FUNCTION_BLOCK fb_eventController
VAR_INPUT
in_flg_run : BOOL;
END_VAR
VAR_OUTPUT
	out_flg_run : BOOL;
END_VAR
VAR

	fbi_eventListGenerator: ARRAY [0..50] OF fb_eventListGenerator;
	var_semaphore: INT;
	var_alarmQty: INT;
	flg_errorTrg: ARRAY[0..50] OF BOOL;

    var_timeAsDT : DT;
	var_alarmListLog: s_alarmList;
	flg_reqUpdate: BOOL;
	fbi_r_TRIG: R_TRIG;
	var_n: INT;
	fbi_buzzerGenerater: fb_buzzerGenerater;
	var_n2: INT;
	var_alarmListEmpty : s_alarmList;
	fbi_GetLocalAmsNetId: FB_GetLocalAmsNetId;
	fbi_LocalSystemTime: FB_LocalSystemTime;
	fbi_ton1: TON;
	var_i: INT;
	fbi_first: TON;
	var_dummy: ARRAY [1..10] OF s_str_alarmList;
END_VAR
VAR_STAT
	flg_error: BOOL;
	flg_warning: BOOL;
	flg_info: BOOL;
END_VAR
VAR // added by the converter: edge detectors and wires of the graphical bodies
    _rt1 : R_TRIG;
END_VAR

eventList();

//get current time
fbi_GetLocalAmsNetId(
	bExecute:=TRUE , 
	tTimeOut:= ,
	bBusy=> , 
	bError=> , 
	nErrId=> , 
	AddrString=> , 
	AddrBytes=> );


fbi_LocalSystemTime(
	sNetID:=fbi_GetLocalAmsNetId.AddrString , 
	bEnable:= TRUE, 
	dwCycle:= , 
	dwOpt:= , 
	tTimeout:= , 
	bValid=> , 
	systemTime=> , 
	tzID=> );

var_timeAsDT := SYSTEMTIME_TO_DT(fbi_LocalSystemTime.systemTime);
//reset

//
IF gvl_error.flg_error THEN
	gvl_error.flg_alramBusy := TRUE;
END_IF

fbi_r_TRIG(CLK:= flg_requpdate, Q=> );
//event log update
IF fbi_r_TRIG.Q THEN
	FOR var_n := 50 TO 2 BY -1 DO
			gvl_error.var_ary_alarmlistLog[var_n].var_alarmName := gvl_error.var_ary_alarmlistLog[var_n-1].var_alarmName;
			gvl_error.var_ary_alarmlistLog[var_n].var_alarmLevel := gvl_error.var_ary_alarmlistLog[var_n-1].var_alarmLevel;
			gvl_error.var_ary_alarmlistLog[var_n].var_alarmMassge := gvl_error.var_ary_alarmlistLog[var_n-1].var_alarmMassge;
			gvl_error.var_ary_alarmlistLog[var_n].var_alarmTime := gvl_error.var_ary_alarmlistLog[var_n-1].var_alarmTime;
			gvl_error.var_ary_alarmlistLog[var_n].var_alarmCode1 := gvl_error.var_ary_alarmlistLog[var_n-1].var_alarmCode1;
			gvl_error.var_ary_alarmlistLog[var_n].var_alarmCode2 := gvl_error.var_ary_alarmlistLog[var_n-1].var_alarmCode2;
			
			IF var_n = 2 THEN
				gvl_error.var_ary_alarmlistLog[1].var_alarmName := var_alarmListLog.var_alarmName;
				gvl_error.var_ary_alarmlistLog[1].var_alarmLevel := var_alarmListLog.var_alarmLevel;
				gvl_error.var_ary_alarmlistLog[1].var_alarmMassge := var_alarmListLog.var_alarmMassge;
				gvl_error.var_ary_alarmlistLog[1].var_alarmTime := var_alarmListLog.var_alarmTime;
				gvl_error.var_ary_alarmlistLog[1].var_alarmCode1 := var_alarmListLog.var_alarmCode1;
				gvl_error.var_ary_alarmlistLog[1].var_alarmCode2 := var_alarmListLog.var_alarmCode2;
				var_semaphore := var_semaphore - 1;
			END_IF
		END_FOR	
END_IF

//reset realtime event 
IF gvl_error.flg_eventDisplayRest THEN
	FOR var_n2 := 1 TO 10 BY 1 DO
		gvl_error.var_ary_alarmlistActive[var_n2].var_alarmCode1 := eP_alarmCode._;
		gvl_error.var_ary_alarmlistActive[var_n2].var_alarmCode2 := '';
		gvl_error.var_ary_alarmlistActive[var_n2].var_alarmLevel := '';
		gvl_error.var_ary_alarmlistActive[var_n2].var_alarmMassge := "";
		gvl_error.var_ary_alarmlistActive[var_n2].var_alarmName := "";
		gvl_error.var_ary_alarmlistActive[var_n2].var_alarmTime := '';
	END_FOR
END_IF
//massage
	flg_info := gvl_error.flg_warning OR gvl_error.flg_info OR gvl_error.flg_sample_windown_warning;
	IF NOT flg_info THEN
		gvl_visu.var_msg := "";	
	END_IF
//buzzer
fbi_buzzerGenerater(
	in_flg_LvError:=gvl_error.flg_error OR gvl_error.flg_sample_windown_warning,
	in_flg_LvWarning:=gvl_error.flg_warning,
	in_flg_LvInfo:=gvl_error.flg_info ,
	out_flg_buzzer=> gvl_io.flg_signalTowerBuzzer ,
	out_flg_Yellow=> gvl_io.flg_signalTowerYellow
);
gvl_io.flg_signalTowerRed := gvl_error.flg_error;

IF gvl_error.flg_ararmLevelRest THEN
	gvl_error.flg_error := FALSE;
	gvl_error.flg_warning := FALSE;
	gvl_error.flg_info := FALSE;
END_IF

ACTION eventList:
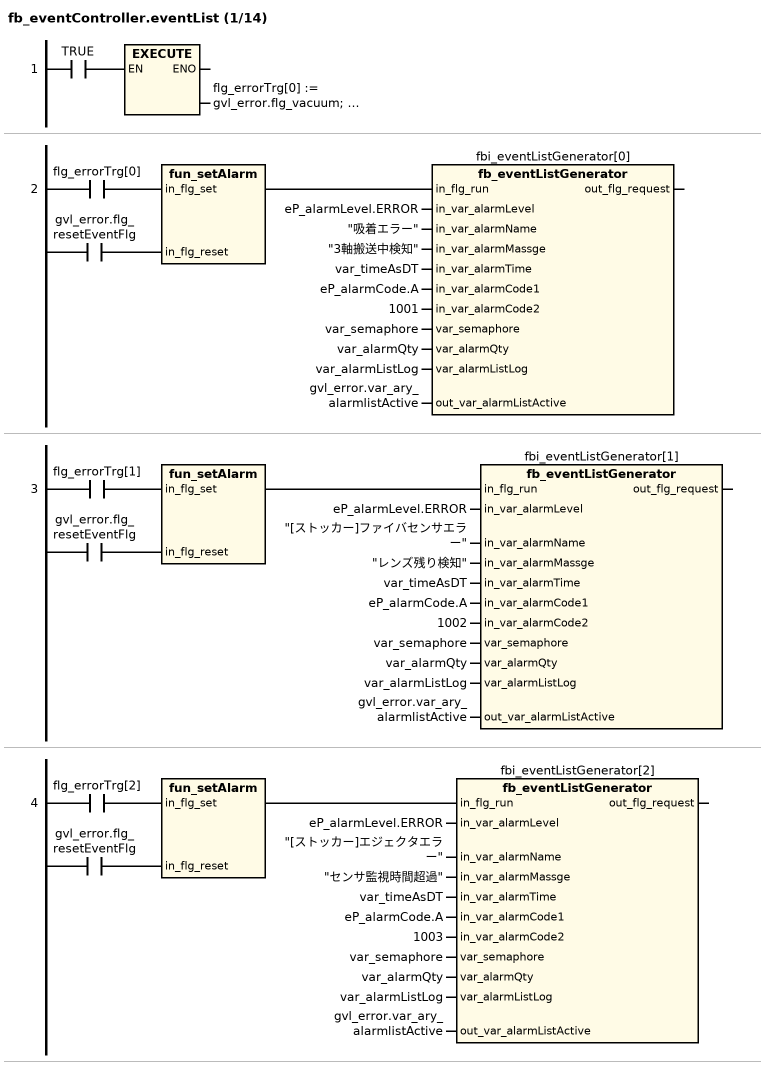
// NETWORK 1
flg_errorTrg[0] := gvl_error.flg_vacuum;
flg_errorTrg[1] := gvl_error.flg_fiberSens;
flg_errorTrg[2] := gvl_solv.fbi_ejector.out_flg_error;
flg_errorTrg[3] := gvl_solv.fbi_chuck.out_flg_error;
flg_errorTrg[4] := gvl_solv.fbi_push.out_flg_error;
flg_errorTrg[5] := gvl_elecylinder.fbi_axisTransport.out_flg_error;
flg_errorTrg[6] := gvl_elecylinder.fbi_axisSample.out_flg_error;
flg_errorTrg[7] := gvl_elecylinder.fbi_axisTrayChange.out_flg_error OR gvl_error.flg_trayChangeError;
flg_errorTrg[8] := gvl_elecylinder.ref_axis_transport.input.in_wire_error;
flg_errorTrg[9] := gvl_elecylinder.ref_axis_sample.input.in_wire_error;
flg_errorTrg[10] := gvl_elecylinder.ref_axis_trayChange.input.in_wire_error;
flg_errorTrg[11] := gvl_axis.ref_x.Error;
flg_errorTrg[12] := gvl_axis.ref_y.Error;
flg_errorTrg[13] := gvl_axis.ref_z.Error;
flg_errorTrg[14] := gvl_elecylinder.fbi_axisRotary.out_flg_error;
flg_errorTrg[15] := gvl_elecylinder.ref_axis_rotary.input.in_wire_error;
flg_errorTrg[16] := NOT gvl_io.flg_saftyUnitState;
flg_errorTrg[17] := NOT gvl_io.flg_frontSaftyDoor;
flg_errorTrg[18] := gvl_io.flg_gatemeasurementStatus;
flg_errorTrg[19] := gvl_axis.fbi_mc_jogX.Error;
flg_errorTrg[20] := gvl_axis.fbi_mc_jogY.Error;
flg_errorTrg[21] := gvl_axis.fbi_mc_jogZ.Error;
flg_errorTrg[22] := gvl_auto.flg_trayChangeDone OR NOT  gvl_visu.flg_btn_trayChangeDone ;
flg_errorTrg[23] := gvl_error.flg_gm_fiberSens; 
flg_errorTrg[24] := gvl_solv.fbi_gm_ejector.out_flg_error;
flg_errorTrg[25] := gvl_solv.fbi_gm_chuck.out_flg_error;
flg_errorTrg[26] := gvl_solv.fbi_gm_push.out_flg_error;
flg_errorTrg[27] := gvl_elecylinder.fbi_gm_axisPickUp.out_flg_error;
flg_errorTrg[28] := gvl_elecylinder.fbi_gm_axisTransport.out_flg_error;
flg_errorTrg[29] := gvl_axis.ref_r.Error;
flg_errorTrg[30] := gvl_axis.fbi_mc_jogR.Error;
flg_errorTrg[31] := gvl_error.flg_axisXTorqueOver;
flg_errorTrg[32] := gvl_error.flg_axisYTorqueOver;
flg_errorTrg[33] := gvl_error.flg_axisZTorqueOver;
flg_errorTrg[34] := gvl_error.flg_axisRTorqueOver;
flg_errorTrg[35] := gvl_solv.fbi_gm_rotary.out_flg_error;
flg_errorTrg[36] := gvl_solv.fbi_gm_pickup.out_flg_error;
flg_errorTrg[37] := gvl_solv.fbi_gm_stamp.out_flg_error;
flg_errorTrg[38] := gvl_gm.var_incjetInfo.flg_error;
flg_errorTrg[39] := gvl_error.flg_incjet;
flg_errorTrg[40] := gvl_error.flg_sample_windown_error;
//flg_errorTrg[41] := ;
//flg_errorTrg[42] := ;
//flg_errorTrg[43] := ;
//flg_errorTrg[44] := ;
//flg_errorTrg[45] := ;
//flg_errorTrg[46] := ;
//flg_errorTrg[47] := ;
//flg_errorTrg[48] := ;
//flg_errorTrg[49] := ;
//flg_errorTrg[50] := ;

// NETWORK 2
fbi_eventListGenerator[0](
    in_flg_run := fun_setAlarm(in_flg_set := flg_errorTrg[0], in_flg_reset := gvl_error.flg_resetEventFlg),
    in_var_alarmLevel := eP_alarmLevel.ERROR,
    in_var_alarmName := "吸着エラー",
    in_var_alarmMassge := "3軸搬送中検知",
    in_var_alarmTime := var_timeAsDT,
    in_var_alarmCode1 := eP_alarmCode.A,
    in_var_alarmCode2 := 1001,
    var_semaphore := var_semaphore,
    var_alarmQty := var_alarmQty,
    var_alarmListLog := var_alarmListLog,
    out_var_alarmListActive := gvl_error.var_ary_alarmlistActive); // fb_eventListGenerator

// NETWORK 3
fbi_eventListGenerator[1](
    in_flg_run := fun_setAlarm(in_flg_set := flg_errorTrg[1], in_flg_reset := gvl_error.flg_resetEventFlg),
    in_var_alarmLevel := eP_alarmLevel.ERROR,
    in_var_alarmName := "[ストッカー]ファイバセンサエラー",
    in_var_alarmMassge := "レンズ残り検知",
    in_var_alarmTime := var_timeAsDT,
    in_var_alarmCode1 := eP_alarmCode.A,
    in_var_alarmCode2 := 1002,
    var_semaphore := var_semaphore,
    var_alarmQty := var_alarmQty,
    var_alarmListLog := var_alarmListLog,
    out_var_alarmListActive := gvl_error.var_ary_alarmlistActive); // fb_eventListGenerator

// NETWORK 4
fbi_eventListGenerator[2](
    in_flg_run := fun_setAlarm(in_flg_set := flg_errorTrg[2], in_flg_reset := gvl_error.flg_resetEventFlg),
    in_var_alarmLevel := eP_alarmLevel.ERROR,
    in_var_alarmName := "[ストッカー]エジェクタエラー",
    in_var_alarmMassge := "センサ監視時間超過",
    in_var_alarmTime := var_timeAsDT,
    in_var_alarmCode1 := eP_alarmCode.A,
    in_var_alarmCode2 := 1003,
    var_semaphore := var_semaphore,
    var_alarmQty := var_alarmQty,
    var_alarmListLog := var_alarmListLog,
    out_var_alarmListActive := gvl_error.var_ary_alarmlistActive); // fb_eventListGenerator

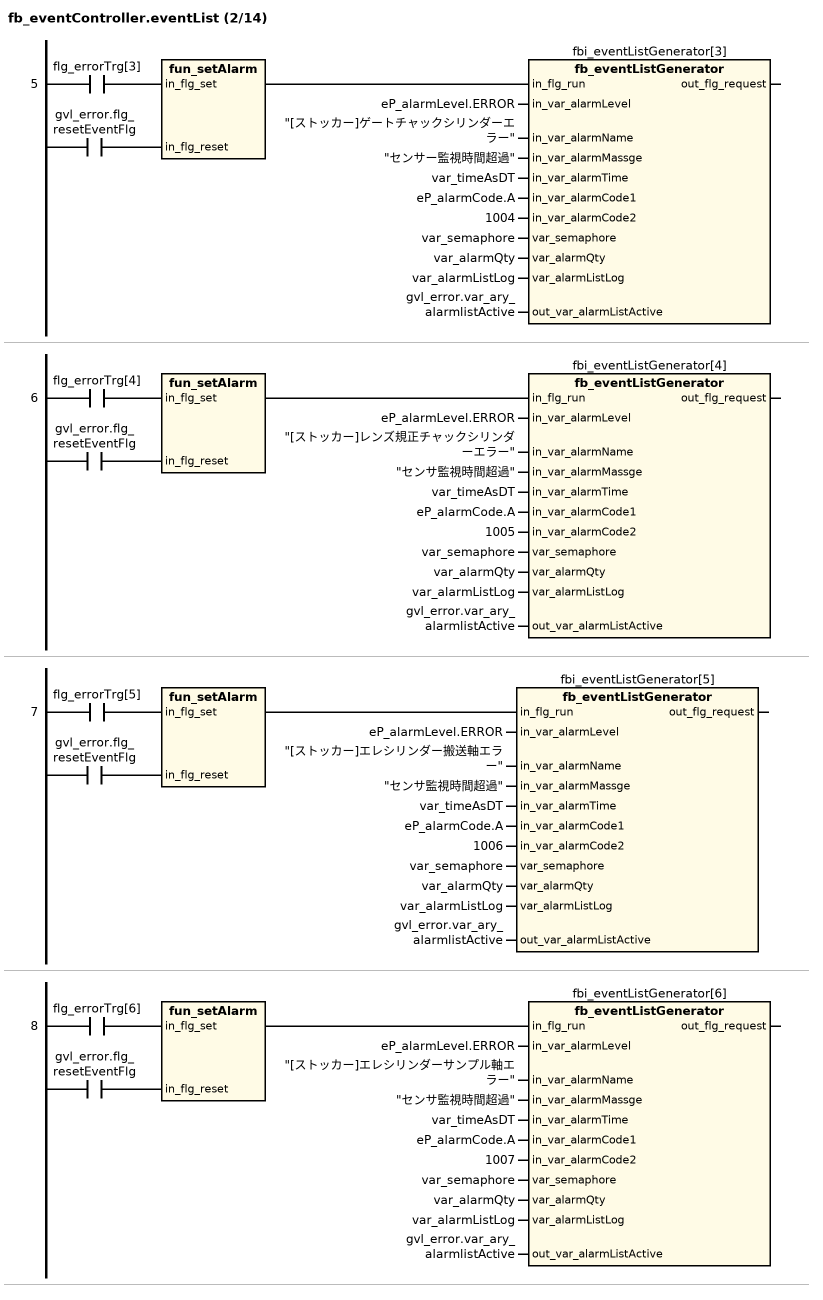
// NETWORK 5
fbi_eventListGenerator[3](
    in_flg_run := fun_setAlarm(in_flg_set := flg_errorTrg[3], in_flg_reset := gvl_error.flg_resetEventFlg),
    in_var_alarmLevel := eP_alarmLevel.ERROR,
    in_var_alarmName := "[ストッカー]ゲートチャックシリンダーエラー",
    in_var_alarmMassge := "センサー監視時間超過",
    in_var_alarmTime := var_timeAsDT,
    in_var_alarmCode1 := eP_alarmCode.A,
    in_var_alarmCode2 := 1004,
    var_semaphore := var_semaphore,
    var_alarmQty := var_alarmQty,
    var_alarmListLog := var_alarmListLog,
    out_var_alarmListActive := gvl_error.var_ary_alarmlistActive); // fb_eventListGenerator

// NETWORK 6
fbi_eventListGenerator[4](
    in_flg_run := fun_setAlarm(in_flg_set := flg_errorTrg[4], in_flg_reset := gvl_error.flg_resetEventFlg),
    in_var_alarmLevel := eP_alarmLevel.ERROR,
    in_var_alarmName := "[ストッカー]レンズ規正チャックシリンダーエラー",
    in_var_alarmMassge := "センサ監視時間超過",
    in_var_alarmTime := var_timeAsDT,
    in_var_alarmCode1 := eP_alarmCode.A,
    in_var_alarmCode2 := 1005,
    var_semaphore := var_semaphore,
    var_alarmQty := var_alarmQty,
    var_alarmListLog := var_alarmListLog,
    out_var_alarmListActive := gvl_error.var_ary_alarmlistActive); // fb_eventListGenerator

// NETWORK 7
fbi_eventListGenerator[5](
    in_flg_run := fun_setAlarm(in_flg_set := flg_errorTrg[5], in_flg_reset := gvl_error.flg_resetEventFlg),
    in_var_alarmLevel := eP_alarmLevel.ERROR,
    in_var_alarmName := "[ストッカー]エレシリンダー搬送軸エラー",
    in_var_alarmMassge := "センサ監視時間超過",
    in_var_alarmTime := var_timeAsDT,
    in_var_alarmCode1 := eP_alarmCode.A,
    in_var_alarmCode2 := 1006,
    var_semaphore := var_semaphore,
    var_alarmQty := var_alarmQty,
    var_alarmListLog := var_alarmListLog,
    out_var_alarmListActive := gvl_error.var_ary_alarmlistActive); // fb_eventListGenerator

// NETWORK 8
fbi_eventListGenerator[6](
    in_flg_run := fun_setAlarm(in_flg_set := flg_errorTrg[6], in_flg_reset := gvl_error.flg_resetEventFlg),
    in_var_alarmLevel := eP_alarmLevel.ERROR,
    in_var_alarmName := "[ストッカー]エレシリンダーサンプル軸エラー",
    in_var_alarmMassge := "センサ監視時間超過",
    in_var_alarmTime := var_timeAsDT,
    in_var_alarmCode1 := eP_alarmCode.A,
    in_var_alarmCode2 := 1007,
    var_semaphore := var_semaphore,
    var_alarmQty := var_alarmQty,
    var_alarmListLog := var_alarmListLog,
    out_var_alarmListActive := gvl_error.var_ary_alarmlistActive); // fb_eventListGenerator

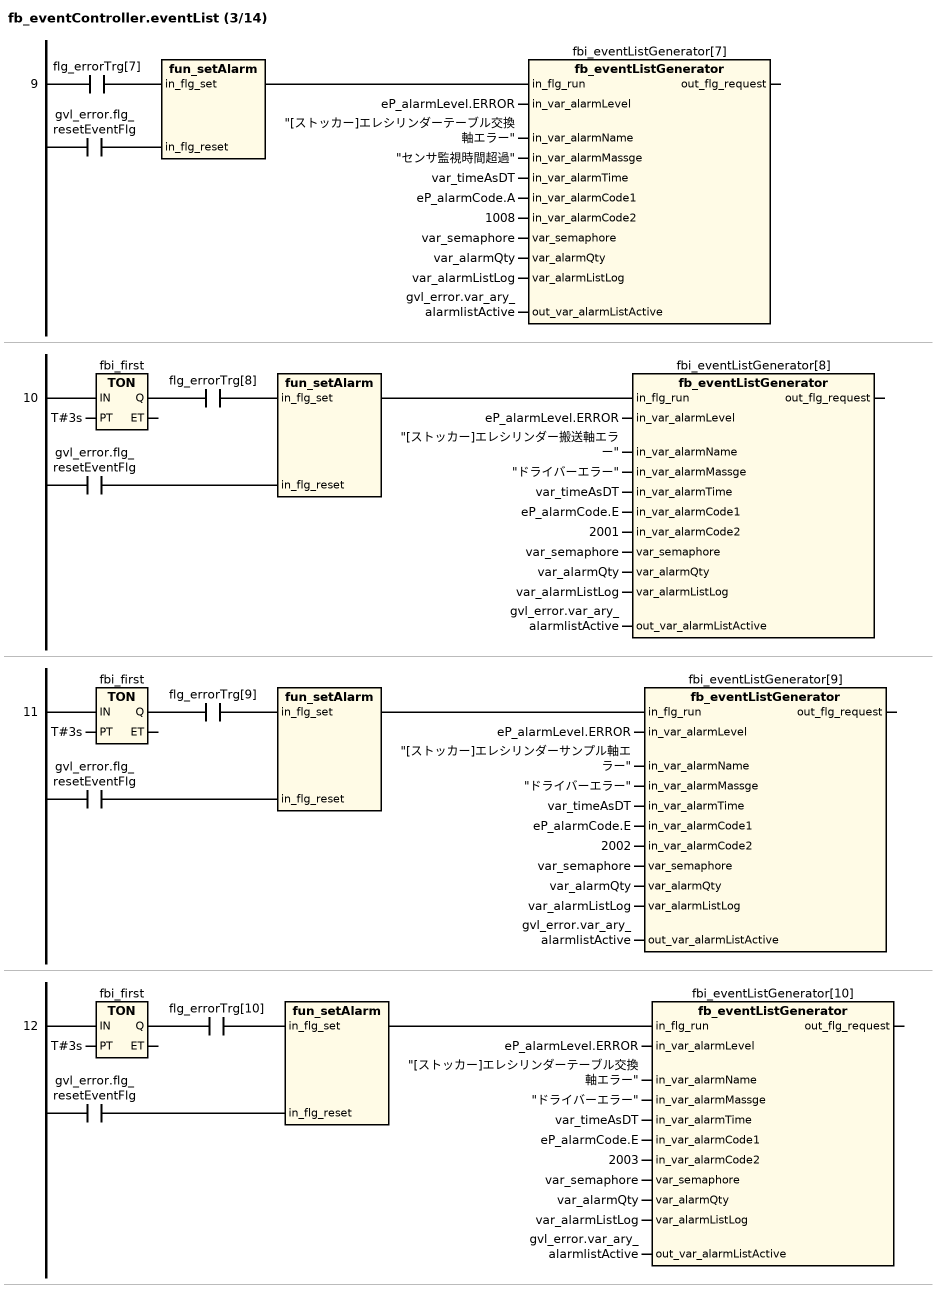
// NETWORK 9
fbi_eventListGenerator[7](
    in_flg_run := fun_setAlarm(in_flg_set := flg_errorTrg[7], in_flg_reset := gvl_error.flg_resetEventFlg),
    in_var_alarmLevel := eP_alarmLevel.ERROR,
    in_var_alarmName := "[ストッカー]エレシリンダーテーブル交換軸エラー",
    in_var_alarmMassge := "センサ監視時間超過",
    in_var_alarmTime := var_timeAsDT,
    in_var_alarmCode1 := eP_alarmCode.A,
    in_var_alarmCode2 := 1008,
    var_semaphore := var_semaphore,
    var_alarmQty := var_alarmQty,
    var_alarmListLog := var_alarmListLog,
    out_var_alarmListActive := gvl_error.var_ary_alarmlistActive); // fb_eventListGenerator

// NETWORK 10
fbi_first(IN := TRUE, PT := T#3s); // TON
fbi_eventListGenerator[8](
    in_flg_run := fun_setAlarm(in_flg_set := fbi_first.Q AND flg_errorTrg[8], in_flg_reset := gvl_error.flg_resetEventFlg),
    in_var_alarmLevel := eP_alarmLevel.ERROR,
    in_var_alarmName := "[ストッカー]エレシリンダー搬送軸エラー",
    in_var_alarmMassge := "ドライバーエラー",
    in_var_alarmTime := var_timeAsDT,
    in_var_alarmCode1 := eP_alarmCode.E,
    in_var_alarmCode2 := 2001,
    var_semaphore := var_semaphore,
    var_alarmQty := var_alarmQty,
    var_alarmListLog := var_alarmListLog,
    out_var_alarmListActive := gvl_error.var_ary_alarmlistActive); // fb_eventListGenerator

// NETWORK 11
fbi_first(IN := TRUE, PT := T#3s); // TON
fbi_eventListGenerator[9](
    in_flg_run := fun_setAlarm(in_flg_set := fbi_first.Q AND flg_errorTrg[9], in_flg_reset := gvl_error.flg_resetEventFlg),
    in_var_alarmLevel := eP_alarmLevel.ERROR,
    in_var_alarmName := "[ストッカー]エレシリンダーサンプル軸エラー",
    in_var_alarmMassge := "ドライバーエラー",
    in_var_alarmTime := var_timeAsDT,
    in_var_alarmCode1 := eP_alarmCode.E,
    in_var_alarmCode2 := 2002,
    var_semaphore := var_semaphore,
    var_alarmQty := var_alarmQty,
    var_alarmListLog := var_alarmListLog,
    out_var_alarmListActive := gvl_error.var_ary_alarmlistActive); // fb_eventListGenerator

// NETWORK 12
fbi_first(IN := TRUE, PT := T#3s); // TON
fbi_eventListGenerator[10](
    in_flg_run := fun_setAlarm(in_flg_set := fbi_first.Q AND flg_errorTrg[10], in_flg_reset := gvl_error.flg_resetEventFlg),
    in_var_alarmLevel := eP_alarmLevel.ERROR,
    in_var_alarmName := "[ストッカー]エレシリンダーテーブル交換軸エラー",
    in_var_alarmMassge := "ドライバーエラー",
    in_var_alarmTime := var_timeAsDT,
    in_var_alarmCode1 := eP_alarmCode.E,
    in_var_alarmCode2 := 2003,
    var_semaphore := var_semaphore,
    var_alarmQty := var_alarmQty,
    var_alarmListLog := var_alarmListLog,
    out_var_alarmListActive := gvl_error.var_ary_alarmlistActive); // fb_eventListGenerator

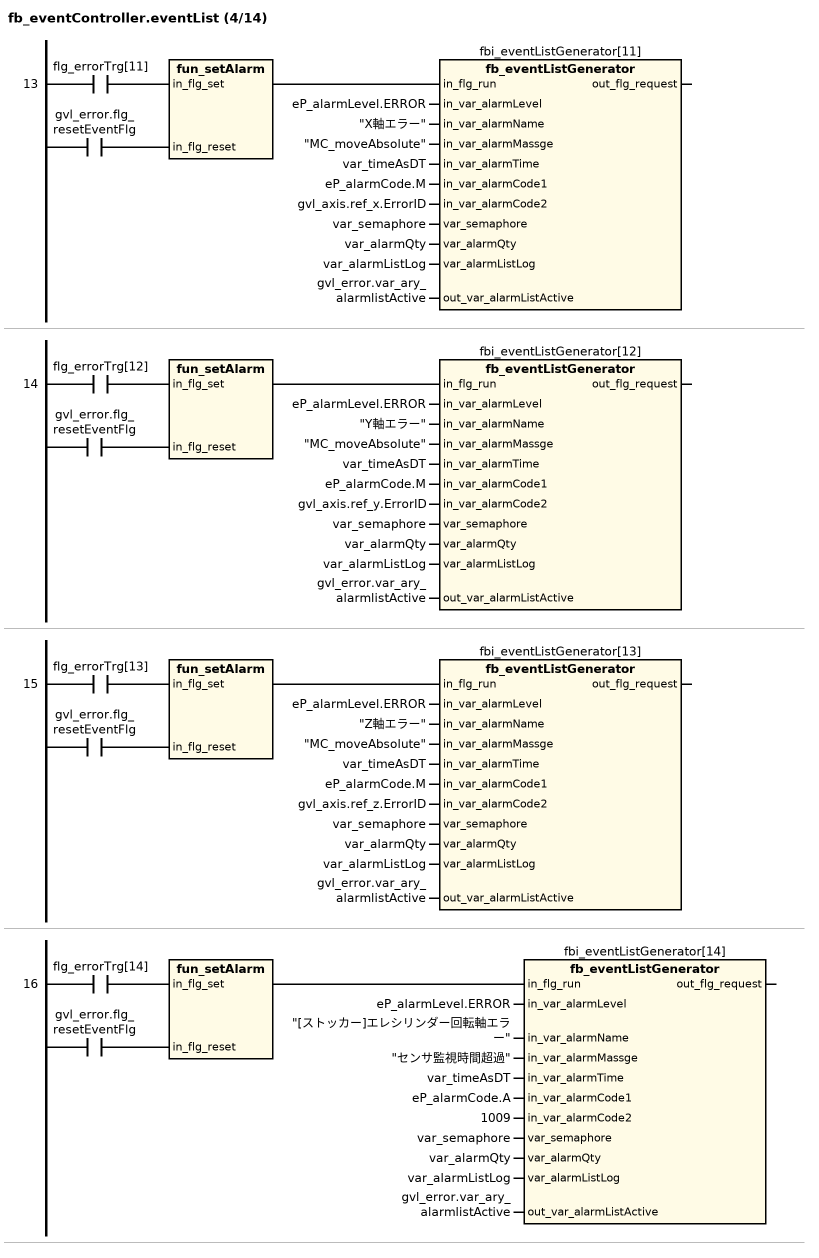
// NETWORK 13
fbi_eventListGenerator[11](
    in_flg_run := fun_setAlarm(in_flg_set := flg_errorTrg[11], in_flg_reset := gvl_error.flg_resetEventFlg),
    in_var_alarmLevel := eP_alarmLevel.ERROR,
    in_var_alarmName := "X軸エラー",
    in_var_alarmMassge := "MC_moveAbsolute",
    in_var_alarmTime := var_timeAsDT,
    in_var_alarmCode1 := eP_alarmCode.M,
    in_var_alarmCode2 := gvl_axis.ref_x.ErrorID,
    var_semaphore := var_semaphore,
    var_alarmQty := var_alarmQty,
    var_alarmListLog := var_alarmListLog,
    out_var_alarmListActive := gvl_error.var_ary_alarmlistActive); // fb_eventListGenerator

// NETWORK 14
fbi_eventListGenerator[12](
    in_flg_run := fun_setAlarm(in_flg_set := flg_errorTrg[12], in_flg_reset := gvl_error.flg_resetEventFlg),
    in_var_alarmLevel := eP_alarmLevel.ERROR,
    in_var_alarmName := "Y軸エラー",
    in_var_alarmMassge := "MC_moveAbsolute",
    in_var_alarmTime := var_timeAsDT,
    in_var_alarmCode1 := eP_alarmCode.M,
    in_var_alarmCode2 := gvl_axis.ref_y.ErrorID,
    var_semaphore := var_semaphore,
    var_alarmQty := var_alarmQty,
    var_alarmListLog := var_alarmListLog,
    out_var_alarmListActive := gvl_error.var_ary_alarmlistActive); // fb_eventListGenerator

// NETWORK 15
fbi_eventListGenerator[13](
    in_flg_run := fun_setAlarm(in_flg_set := flg_errorTrg[13], in_flg_reset := gvl_error.flg_resetEventFlg),
    in_var_alarmLevel := eP_alarmLevel.ERROR,
    in_var_alarmName := "Z軸エラー",
    in_var_alarmMassge := "MC_moveAbsolute",
    in_var_alarmTime := var_timeAsDT,
    in_var_alarmCode1 := eP_alarmCode.M,
    in_var_alarmCode2 := gvl_axis.ref_z.ErrorID,
    var_semaphore := var_semaphore,
    var_alarmQty := var_alarmQty,
    var_alarmListLog := var_alarmListLog,
    out_var_alarmListActive := gvl_error.var_ary_alarmlistActive); // fb_eventListGenerator

// NETWORK 16
fbi_eventListGenerator[14](
    in_flg_run := fun_setAlarm(in_flg_set := flg_errorTrg[14], in_flg_reset := gvl_error.flg_resetEventFlg),
    in_var_alarmLevel := eP_alarmLevel.ERROR,
    in_var_alarmName := "[ストッカー]エレシリンダー回転軸エラー",
    in_var_alarmMassge := "センサ監視時間超過",
    in_var_alarmTime := var_timeAsDT,
    in_var_alarmCode1 := eP_alarmCode.A,
    in_var_alarmCode2 := 1009,
    var_semaphore := var_semaphore,
    var_alarmQty := var_alarmQty,
    var_alarmListLog := var_alarmListLog,
    out_var_alarmListActive := gvl_error.var_ary_alarmlistActive); // fb_eventListGenerator

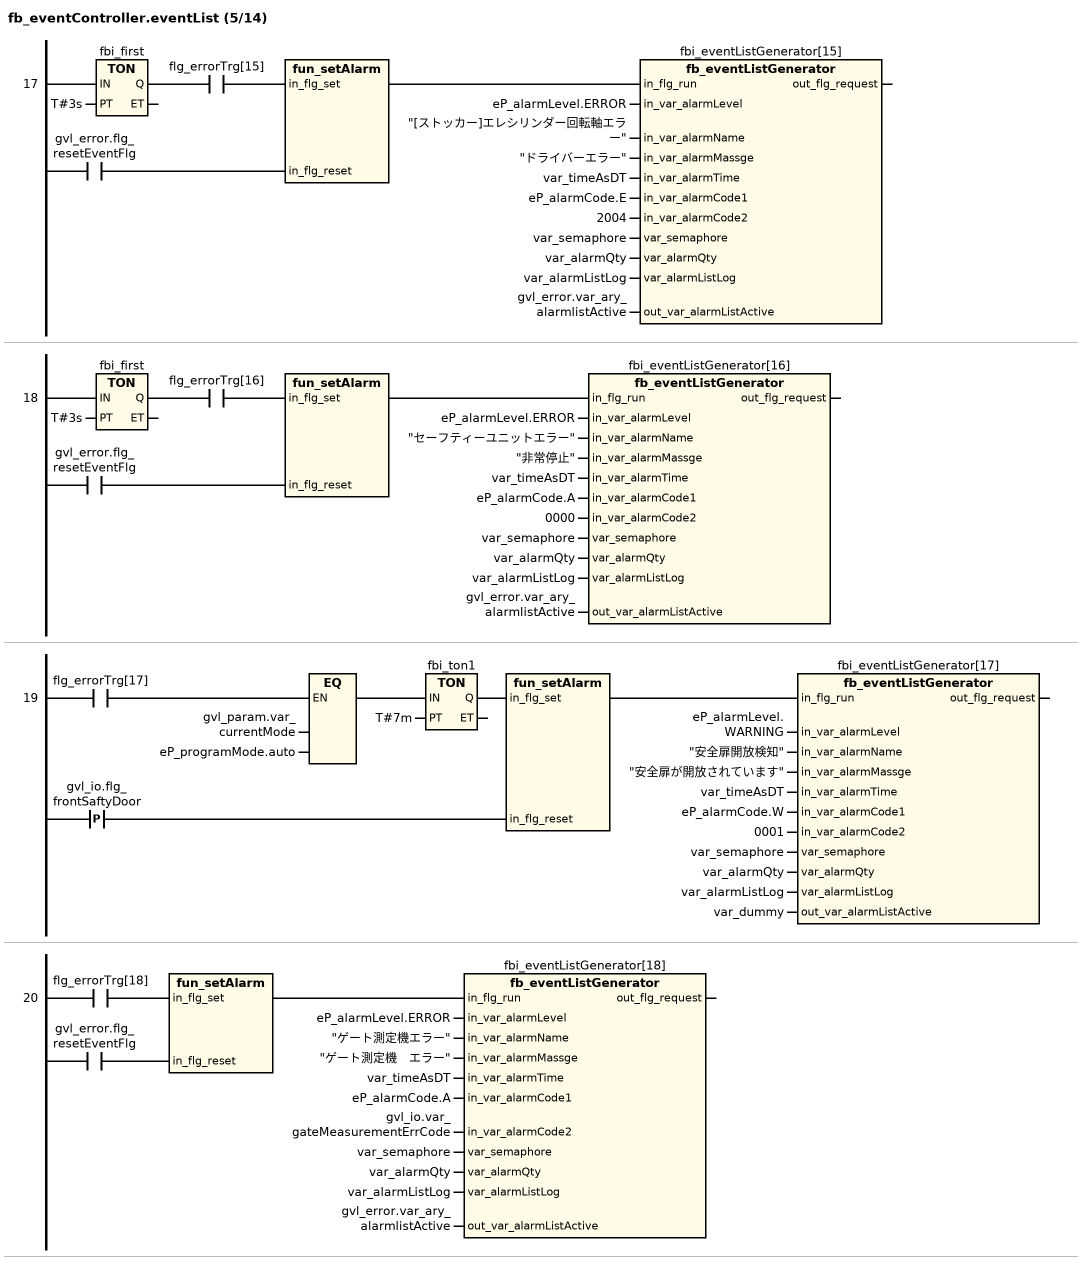
// NETWORK 17
fbi_first(IN := TRUE, PT := T#3s); // TON
fbi_eventListGenerator[15](
    in_flg_run := fun_setAlarm(in_flg_set := fbi_first.Q AND flg_errorTrg[15], in_flg_reset := gvl_error.flg_resetEventFlg),
    in_var_alarmLevel := eP_alarmLevel.ERROR,
    in_var_alarmName := "[ストッカー]エレシリンダー回転軸エラー",
    in_var_alarmMassge := "ドライバーエラー",
    in_var_alarmTime := var_timeAsDT,
    in_var_alarmCode1 := eP_alarmCode.E,
    in_var_alarmCode2 := 2004,
    var_semaphore := var_semaphore,
    var_alarmQty := var_alarmQty,
    var_alarmListLog := var_alarmListLog,
    out_var_alarmListActive := gvl_error.var_ary_alarmlistActive); // fb_eventListGenerator

// NETWORK 18
fbi_first(IN := TRUE, PT := T#3s); // TON
fbi_eventListGenerator[16](
    in_flg_run := fun_setAlarm(in_flg_set := fbi_first.Q AND flg_errorTrg[16], in_flg_reset := gvl_error.flg_resetEventFlg),
    in_var_alarmLevel := eP_alarmLevel.ERROR,
    in_var_alarmName := "セーフティーユニットエラー",
    in_var_alarmMassge := "非常停止",
    in_var_alarmTime := var_timeAsDT,
    in_var_alarmCode1 := eP_alarmCode.A,
    in_var_alarmCode2 := 0000,
    var_semaphore := var_semaphore,
    var_alarmQty := var_alarmQty,
    var_alarmListLog := var_alarmListLog,
    out_var_alarmListActive := gvl_error.var_ary_alarmlistActive); // fb_eventListGenerator

// NETWORK 19
fbi_ton1(IN := flg_errorTrg[17] AND gvl_param.var_currentMode = eP_programMode.auto, PT := T#7m); // TON
_rt1(CLK := gvl_io.flg_frontSaftyDoor);
fbi_eventListGenerator[17](
    in_flg_run := fun_setAlarm(in_flg_set := fbi_ton1.Q, in_flg_reset := _rt1.Q),
    in_var_alarmLevel := eP_alarmLevel.WARNING,
    in_var_alarmName := "安全扉開放検知",
    in_var_alarmMassge := "安全扉が開放されています",
    in_var_alarmTime := var_timeAsDT,
    in_var_alarmCode1 := eP_alarmCode.W,
    in_var_alarmCode2 := 0001,
    var_semaphore := var_semaphore,
    var_alarmQty := var_alarmQty,
    var_alarmListLog := var_alarmListLog,
    out_var_alarmListActive := var_dummy); // fb_eventListGenerator

// NETWORK 20
fbi_eventListGenerator[18](
    in_flg_run := fun_setAlarm(in_flg_set := flg_errorTrg[18], in_flg_reset := gvl_error.flg_resetEventFlg),
    in_var_alarmLevel := eP_alarmLevel.ERROR,
    in_var_alarmName := "ゲート測定機エラー",
    in_var_alarmMassge := "ゲート測定機　エラー",
    in_var_alarmTime := var_timeAsDT,
    in_var_alarmCode1 := eP_alarmCode.A,
    in_var_alarmCode2 := gvl_io.var_gateMeasurementErrCode,
    var_semaphore := var_semaphore,
    var_alarmQty := var_alarmQty,
    var_alarmListLog := var_alarmListLog,
    out_var_alarmListActive := gvl_error.var_ary_alarmlistActive); // fb_eventListGenerator

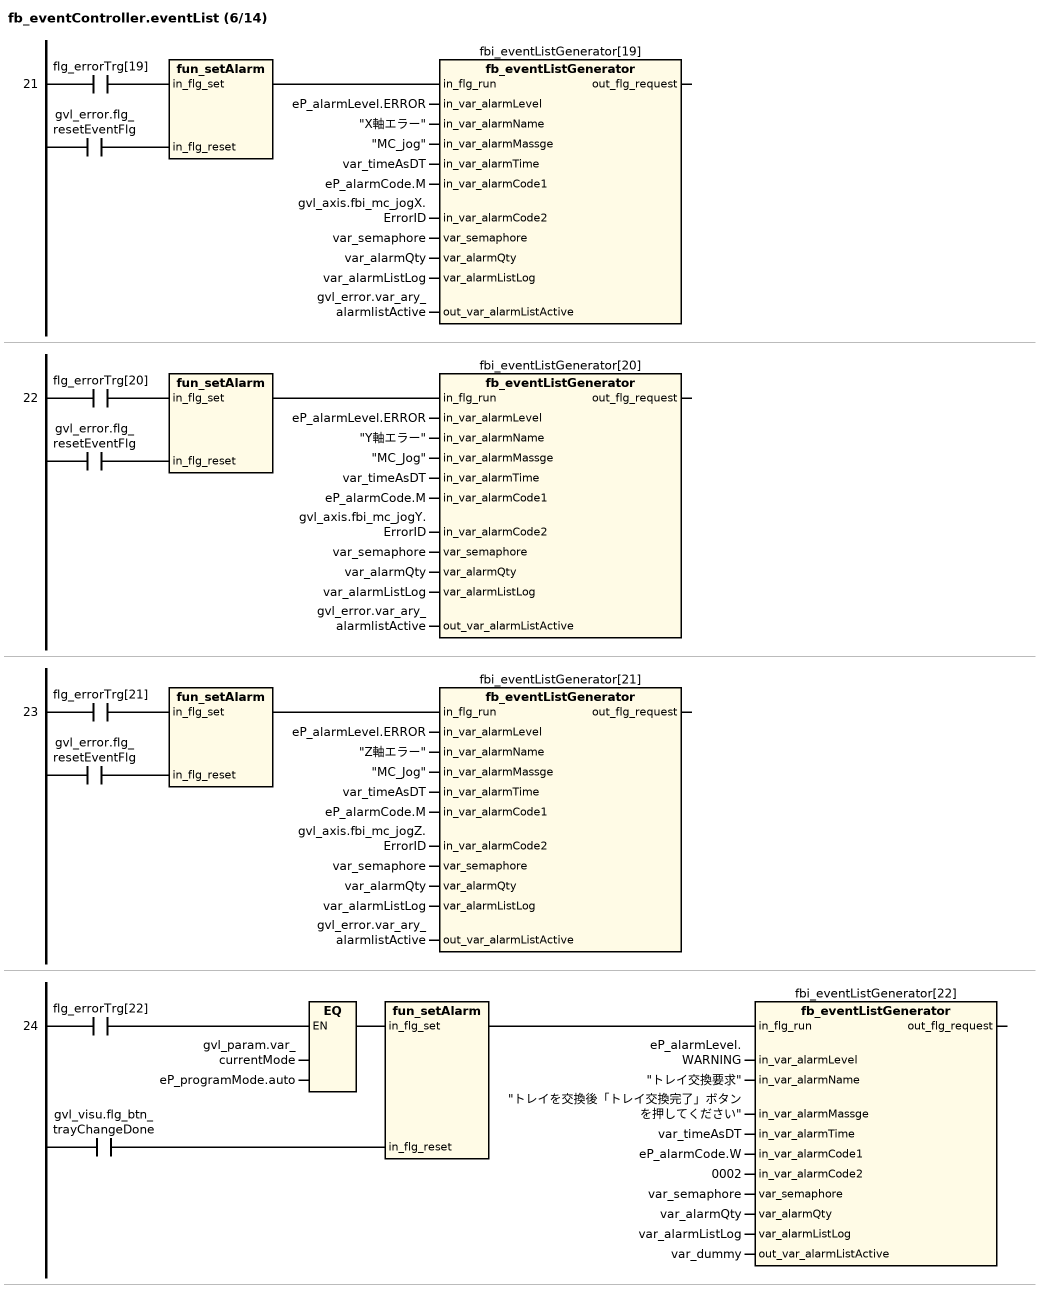
// NETWORK 21
fbi_eventListGenerator[19](
    in_flg_run := fun_setAlarm(in_flg_set := flg_errorTrg[19], in_flg_reset := gvl_error.flg_resetEventFlg),
    in_var_alarmLevel := eP_alarmLevel.ERROR,
    in_var_alarmName := "X軸エラー",
    in_var_alarmMassge := "MC_jog",
    in_var_alarmTime := var_timeAsDT,
    in_var_alarmCode1 := eP_alarmCode.M,
    in_var_alarmCode2 := gvl_axis.fbi_mc_jogX.ErrorID,
    var_semaphore := var_semaphore,
    var_alarmQty := var_alarmQty,
    var_alarmListLog := var_alarmListLog,
    out_var_alarmListActive := gvl_error.var_ary_alarmlistActive); // fb_eventListGenerator

// NETWORK 22
fbi_eventListGenerator[20](
    in_flg_run := fun_setAlarm(in_flg_set := flg_errorTrg[20], in_flg_reset := gvl_error.flg_resetEventFlg),
    in_var_alarmLevel := eP_alarmLevel.ERROR,
    in_var_alarmName := "Y軸エラー",
    in_var_alarmMassge := "MC_Jog",
    in_var_alarmTime := var_timeAsDT,
    in_var_alarmCode1 := eP_alarmCode.M,
    in_var_alarmCode2 := gvl_axis.fbi_mc_jogY.ErrorID,
    var_semaphore := var_semaphore,
    var_alarmQty := var_alarmQty,
    var_alarmListLog := var_alarmListLog,
    out_var_alarmListActive := gvl_error.var_ary_alarmlistActive); // fb_eventListGenerator

// NETWORK 23
fbi_eventListGenerator[21](
    in_flg_run := fun_setAlarm(in_flg_set := flg_errorTrg[21], in_flg_reset := gvl_error.flg_resetEventFlg),
    in_var_alarmLevel := eP_alarmLevel.ERROR,
    in_var_alarmName := "Z軸エラー",
    in_var_alarmMassge := "MC_Jog",
    in_var_alarmTime := var_timeAsDT,
    in_var_alarmCode1 := eP_alarmCode.M,
    in_var_alarmCode2 := gvl_axis.fbi_mc_jogZ.ErrorID,
    var_semaphore := var_semaphore,
    var_alarmQty := var_alarmQty,
    var_alarmListLog := var_alarmListLog,
    out_var_alarmListActive := gvl_error.var_ary_alarmlistActive); // fb_eventListGenerator

// NETWORK 24
fbi_eventListGenerator[22](
    in_flg_run := fun_setAlarm(in_flg_set := flg_errorTrg[22] AND gvl_param.var_currentMode = eP_programMode.auto, in_flg_reset := gvl_visu.flg_btn_trayChangeDone),
    in_var_alarmLevel := eP_alarmLevel.WARNING,
    in_var_alarmName := "トレイ交換要求",
    in_var_alarmMassge := "トレイを交換後「トレイ交換完了」ボタンを押してください",
    in_var_alarmTime := var_timeAsDT,
    in_var_alarmCode1 := eP_alarmCode.W,
    in_var_alarmCode2 := 0002,
    var_semaphore := var_semaphore,
    var_alarmQty := var_alarmQty,
    var_alarmListLog := var_alarmListLog,
    out_var_alarmListActive := var_dummy); // fb_eventListGenerator

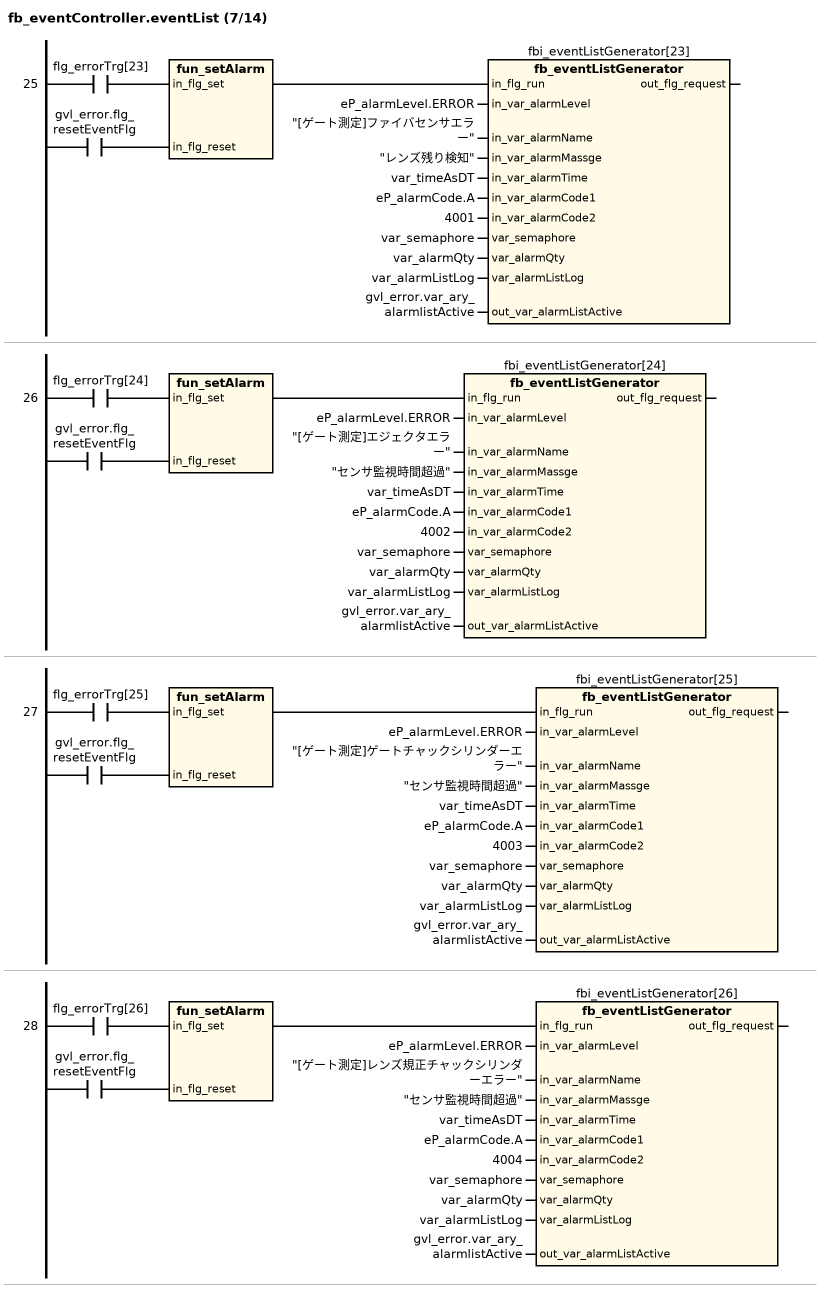
// NETWORK 25
fbi_eventListGenerator[23](
    in_flg_run := fun_setAlarm(in_flg_set := flg_errorTrg[23], in_flg_reset := gvl_error.flg_resetEventFlg),
    in_var_alarmLevel := eP_alarmLevel.ERROR,
    in_var_alarmName := "[ゲート測定]ファイバセンサエラー",
    in_var_alarmMassge := "レンズ残り検知",
    in_var_alarmTime := var_timeAsDT,
    in_var_alarmCode1 := eP_alarmCode.A,
    in_var_alarmCode2 := 4001,
    var_semaphore := var_semaphore,
    var_alarmQty := var_alarmQty,
    var_alarmListLog := var_alarmListLog,
    out_var_alarmListActive := gvl_error.var_ary_alarmlistActive); // fb_eventListGenerator

// NETWORK 26
fbi_eventListGenerator[24](
    in_flg_run := fun_setAlarm(in_flg_set := flg_errorTrg[24], in_flg_reset := gvl_error.flg_resetEventFlg),
    in_var_alarmLevel := eP_alarmLevel.ERROR,
    in_var_alarmName := "[ゲート測定]エジェクタエラー",
    in_var_alarmMassge := "センサ監視時間超過",
    in_var_alarmTime := var_timeAsDT,
    in_var_alarmCode1 := eP_alarmCode.A,
    in_var_alarmCode2 := 4002,
    var_semaphore := var_semaphore,
    var_alarmQty := var_alarmQty,
    var_alarmListLog := var_alarmListLog,
    out_var_alarmListActive := gvl_error.var_ary_alarmlistActive); // fb_eventListGenerator

// NETWORK 27
fbi_eventListGenerator[25](
    in_flg_run := fun_setAlarm(in_flg_set := flg_errorTrg[25], in_flg_reset := gvl_error.flg_resetEventFlg),
    in_var_alarmLevel := eP_alarmLevel.ERROR,
    in_var_alarmName := "[ゲート測定]ゲートチャックシリンダーエラー",
    in_var_alarmMassge := "センサ監視時間超過",
    in_var_alarmTime := var_timeAsDT,
    in_var_alarmCode1 := eP_alarmCode.A,
    in_var_alarmCode2 := 4003,
    var_semaphore := var_semaphore,
    var_alarmQty := var_alarmQty,
    var_alarmListLog := var_alarmListLog,
    out_var_alarmListActive := gvl_error.var_ary_alarmlistActive); // fb_eventListGenerator

// NETWORK 28
fbi_eventListGenerator[26](
    in_flg_run := fun_setAlarm(in_flg_set := flg_errorTrg[26], in_flg_reset := gvl_error.flg_resetEventFlg),
    in_var_alarmLevel := eP_alarmLevel.ERROR,
    in_var_alarmName := "[ゲート測定]レンズ規正チャックシリンダーエラー",
    in_var_alarmMassge := "センサ監視時間超過",
    in_var_alarmTime := var_timeAsDT,
    in_var_alarmCode1 := eP_alarmCode.A,
    in_var_alarmCode2 := 4004,
    var_semaphore := var_semaphore,
    var_alarmQty := var_alarmQty,
    var_alarmListLog := var_alarmListLog,
    out_var_alarmListActive := gvl_error.var_ary_alarmlistActive); // fb_eventListGenerator

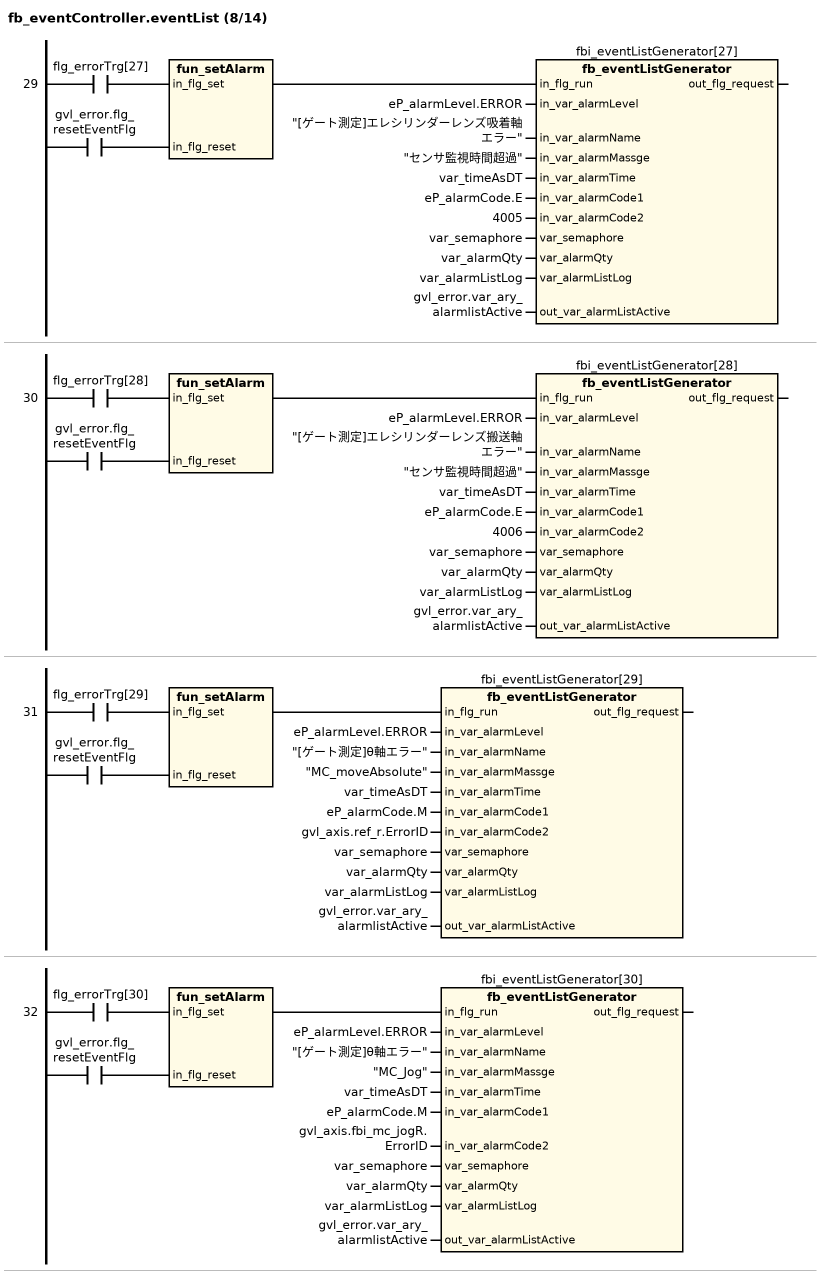
// NETWORK 29
fbi_eventListGenerator[27](
    in_flg_run := fun_setAlarm(in_flg_set := flg_errorTrg[27], in_flg_reset := gvl_error.flg_resetEventFlg),
    in_var_alarmLevel := eP_alarmLevel.ERROR,
    in_var_alarmName := "[ゲート測定]エレシリンダーレンズ吸着軸エラー",
    in_var_alarmMassge := "センサ監視時間超過",
    in_var_alarmTime := var_timeAsDT,
    in_var_alarmCode1 := eP_alarmCode.E,
    in_var_alarmCode2 := 4005,
    var_semaphore := var_semaphore,
    var_alarmQty := var_alarmQty,
    var_alarmListLog := var_alarmListLog,
    out_var_alarmListActive := gvl_error.var_ary_alarmlistActive); // fb_eventListGenerator

// NETWORK 30
fbi_eventListGenerator[28](
    in_flg_run := fun_setAlarm(in_flg_set := flg_errorTrg[28], in_flg_reset := gvl_error.flg_resetEventFlg),
    in_var_alarmLevel := eP_alarmLevel.ERROR,
    in_var_alarmName := "[ゲート測定]エレシリンダーレンズ搬送軸エラー",
    in_var_alarmMassge := "センサ監視時間超過",
    in_var_alarmTime := var_timeAsDT,
    in_var_alarmCode1 := eP_alarmCode.E,
    in_var_alarmCode2 := 4006,
    var_semaphore := var_semaphore,
    var_alarmQty := var_alarmQty,
    var_alarmListLog := var_alarmListLog,
    out_var_alarmListActive := gvl_error.var_ary_alarmlistActive); // fb_eventListGenerator

// NETWORK 31
fbi_eventListGenerator[29](
    in_flg_run := fun_setAlarm(in_flg_set := flg_errorTrg[29], in_flg_reset := gvl_error.flg_resetEventFlg),
    in_var_alarmLevel := eP_alarmLevel.ERROR,
    in_var_alarmName := "[ゲート測定]θ軸エラー",
    in_var_alarmMassge := "MC_moveAbsolute",
    in_var_alarmTime := var_timeAsDT,
    in_var_alarmCode1 := eP_alarmCode.M,
    in_var_alarmCode2 := gvl_axis.ref_r.ErrorID,
    var_semaphore := var_semaphore,
    var_alarmQty := var_alarmQty,
    var_alarmListLog := var_alarmListLog,
    out_var_alarmListActive := gvl_error.var_ary_alarmlistActive); // fb_eventListGenerator

// NETWORK 32
fbi_eventListGenerator[30](
    in_flg_run := fun_setAlarm(in_flg_set := flg_errorTrg[30], in_flg_reset := gvl_error.flg_resetEventFlg),
    in_var_alarmLevel := eP_alarmLevel.ERROR,
    in_var_alarmName := "[ゲート測定]θ軸エラー",
    in_var_alarmMassge := "MC_Jog",
    in_var_alarmTime := var_timeAsDT,
    in_var_alarmCode1 := eP_alarmCode.M,
    in_var_alarmCode2 := gvl_axis.fbi_mc_jogR.ErrorID,
    var_semaphore := var_semaphore,
    var_alarmQty := var_alarmQty,
    var_alarmListLog := var_alarmListLog,
    out_var_alarmListActive := gvl_error.var_ary_alarmlistActive); // fb_eventListGenerator

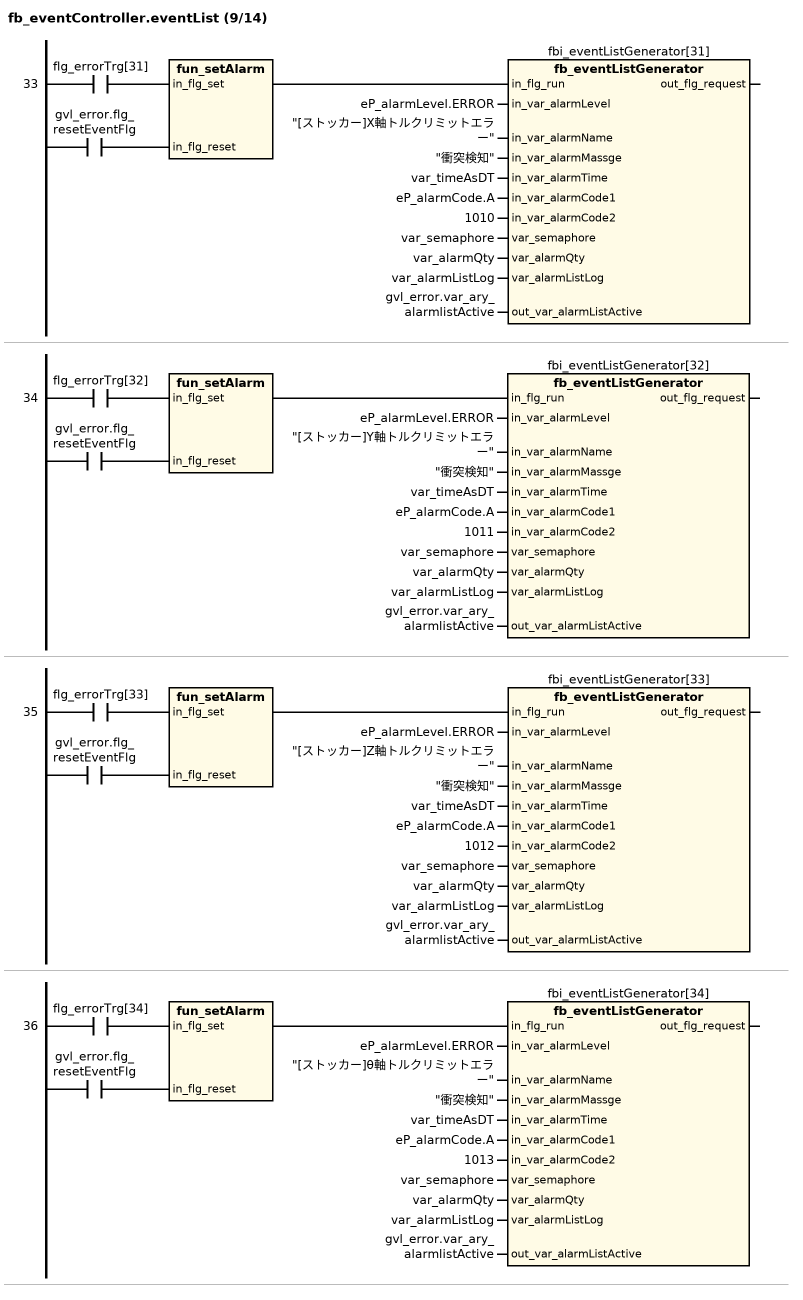
// NETWORK 33
fbi_eventListGenerator[31](
    in_flg_run := fun_setAlarm(in_flg_set := flg_errorTrg[31], in_flg_reset := gvl_error.flg_resetEventFlg),
    in_var_alarmLevel := eP_alarmLevel.ERROR,
    in_var_alarmName := "[ストッカー]X軸トルクリミットエラー",
    in_var_alarmMassge := "衝突検知",
    in_var_alarmTime := var_timeAsDT,
    in_var_alarmCode1 := eP_alarmCode.A,
    in_var_alarmCode2 := 1010,
    var_semaphore := var_semaphore,
    var_alarmQty := var_alarmQty,
    var_alarmListLog := var_alarmListLog,
    out_var_alarmListActive := gvl_error.var_ary_alarmlistActive); // fb_eventListGenerator

// NETWORK 34
fbi_eventListGenerator[32](
    in_flg_run := fun_setAlarm(in_flg_set := flg_errorTrg[32], in_flg_reset := gvl_error.flg_resetEventFlg),
    in_var_alarmLevel := eP_alarmLevel.ERROR,
    in_var_alarmName := "[ストッカー]Y軸トルクリミットエラー",
    in_var_alarmMassge := "衝突検知",
    in_var_alarmTime := var_timeAsDT,
    in_var_alarmCode1 := eP_alarmCode.A,
    in_var_alarmCode2 := 1011,
    var_semaphore := var_semaphore,
    var_alarmQty := var_alarmQty,
    var_alarmListLog := var_alarmListLog,
    out_var_alarmListActive := gvl_error.var_ary_alarmlistActive); // fb_eventListGenerator

// NETWORK 35
fbi_eventListGenerator[33](
    in_flg_run := fun_setAlarm(in_flg_set := flg_errorTrg[33], in_flg_reset := gvl_error.flg_resetEventFlg),
    in_var_alarmLevel := eP_alarmLevel.ERROR,
    in_var_alarmName := "[ストッカー]Z軸トルクリミットエラー",
    in_var_alarmMassge := "衝突検知",
    in_var_alarmTime := var_timeAsDT,
    in_var_alarmCode1 := eP_alarmCode.A,
    in_var_alarmCode2 := 1012,
    var_semaphore := var_semaphore,
    var_alarmQty := var_alarmQty,
    var_alarmListLog := var_alarmListLog,
    out_var_alarmListActive := gvl_error.var_ary_alarmlistActive); // fb_eventListGenerator

// NETWORK 36
fbi_eventListGenerator[34](
    in_flg_run := fun_setAlarm(in_flg_set := flg_errorTrg[34], in_flg_reset := gvl_error.flg_resetEventFlg),
    in_var_alarmLevel := eP_alarmLevel.ERROR,
    in_var_alarmName := "[ストッカー]θ軸トルクリミットエラー",
    in_var_alarmMassge := "衝突検知",
    in_var_alarmTime := var_timeAsDT,
    in_var_alarmCode1 := eP_alarmCode.A,
    in_var_alarmCode2 := 1013,
    var_semaphore := var_semaphore,
    var_alarmQty := var_alarmQty,
    var_alarmListLog := var_alarmListLog,
    out_var_alarmListActive := gvl_error.var_ary_alarmlistActive); // fb_eventListGenerator

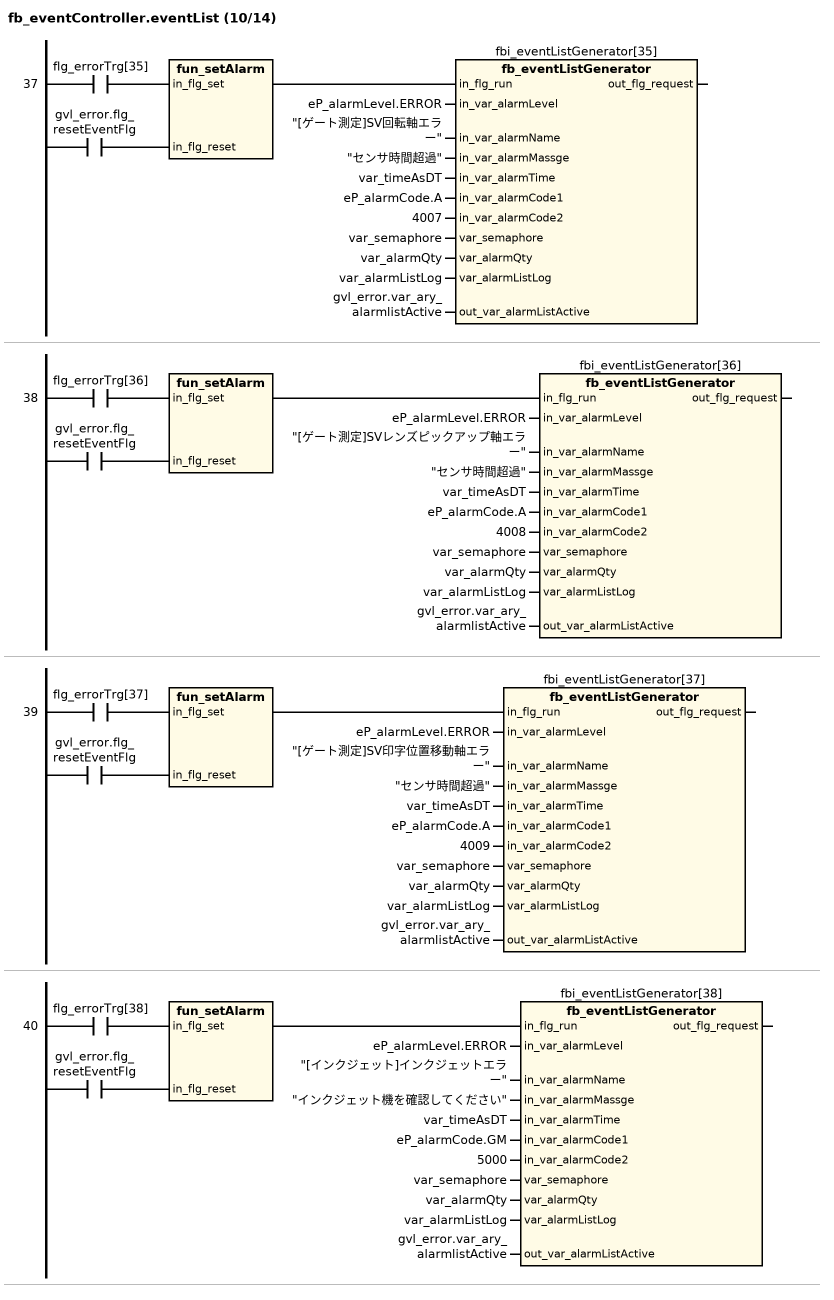
// NETWORK 37
fbi_eventListGenerator[35](
    in_flg_run := fun_setAlarm(in_flg_set := flg_errorTrg[35], in_flg_reset := gvl_error.flg_resetEventFlg),
    in_var_alarmLevel := eP_alarmLevel.ERROR,
    in_var_alarmName := "[ゲート測定]SV回転軸エラー",
    in_var_alarmMassge := "センサ時間超過",
    in_var_alarmTime := var_timeAsDT,
    in_var_alarmCode1 := eP_alarmCode.A,
    in_var_alarmCode2 := 4007,
    var_semaphore := var_semaphore,
    var_alarmQty := var_alarmQty,
    var_alarmListLog := var_alarmListLog,
    out_var_alarmListActive := gvl_error.var_ary_alarmlistActive); // fb_eventListGenerator

// NETWORK 38
fbi_eventListGenerator[36](
    in_flg_run := fun_setAlarm(in_flg_set := flg_errorTrg[36], in_flg_reset := gvl_error.flg_resetEventFlg),
    in_var_alarmLevel := eP_alarmLevel.ERROR,
    in_var_alarmName := "[ゲート測定]SVレンズピックアップ軸エラー",
    in_var_alarmMassge := "センサ時間超過",
    in_var_alarmTime := var_timeAsDT,
    in_var_alarmCode1 := eP_alarmCode.A,
    in_var_alarmCode2 := 4008,
    var_semaphore := var_semaphore,
    var_alarmQty := var_alarmQty,
    var_alarmListLog := var_alarmListLog,
    out_var_alarmListActive := gvl_error.var_ary_alarmlistActive); // fb_eventListGenerator

// NETWORK 39
fbi_eventListGenerator[37](
    in_flg_run := fun_setAlarm(in_flg_set := flg_errorTrg[37], in_flg_reset := gvl_error.flg_resetEventFlg),
    in_var_alarmLevel := eP_alarmLevel.ERROR,
    in_var_alarmName := "[ゲート測定]SV印字位置移動軸エラー",
    in_var_alarmMassge := "センサ時間超過",
    in_var_alarmTime := var_timeAsDT,
    in_var_alarmCode1 := eP_alarmCode.A,
    in_var_alarmCode2 := 4009,
    var_semaphore := var_semaphore,
    var_alarmQty := var_alarmQty,
    var_alarmListLog := var_alarmListLog,
    out_var_alarmListActive := gvl_error.var_ary_alarmlistActive); // fb_eventListGenerator

// NETWORK 40
fbi_eventListGenerator[38](
    in_flg_run := fun_setAlarm(in_flg_set := flg_errorTrg[38], in_flg_reset := gvl_error.flg_resetEventFlg),
    in_var_alarmLevel := eP_alarmLevel.ERROR,
    in_var_alarmName := "[インクジェット]インクジェットエラー",
    in_var_alarmMassge := "インクジェット機を確認してください",
    in_var_alarmTime := var_timeAsDT,
    in_var_alarmCode1 := eP_alarmCode.GM,
    in_var_alarmCode2 := 5000,
    var_semaphore := var_semaphore,
    var_alarmQty := var_alarmQty,
    var_alarmListLog := var_alarmListLog,
    out_var_alarmListActive := gvl_error.var_ary_alarmlistActive); // fb_eventListGenerator

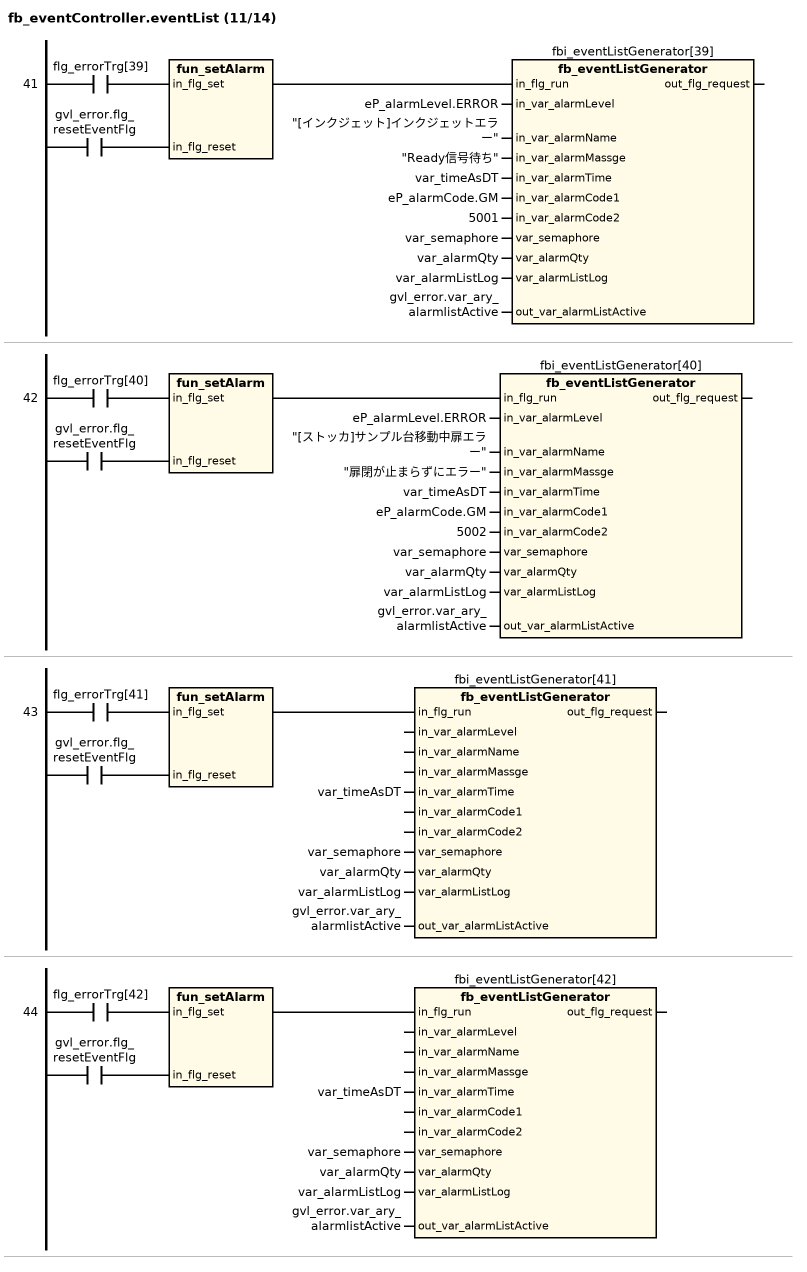
// NETWORK 41
fbi_eventListGenerator[39](
    in_flg_run := fun_setAlarm(in_flg_set := flg_errorTrg[39], in_flg_reset := gvl_error.flg_resetEventFlg),
    in_var_alarmLevel := eP_alarmLevel.ERROR,
    in_var_alarmName := "[インクジェット]インクジェットエラー",
    in_var_alarmMassge := "Ready信号待ち",
    in_var_alarmTime := var_timeAsDT,
    in_var_alarmCode1 := eP_alarmCode.GM,
    in_var_alarmCode2 := 5001,
    var_semaphore := var_semaphore,
    var_alarmQty := var_alarmQty,
    var_alarmListLog := var_alarmListLog,
    out_var_alarmListActive := gvl_error.var_ary_alarmlistActive); // fb_eventListGenerator

// NETWORK 42
fbi_eventListGenerator[40](
    in_flg_run := fun_setAlarm(in_flg_set := flg_errorTrg[40], in_flg_reset := gvl_error.flg_resetEventFlg),
    in_var_alarmLevel := eP_alarmLevel.ERROR,
    in_var_alarmName := "[ストッカ]サンプル台移動中扉エラー",
    in_var_alarmMassge := "扉閉が止まらずにエラー",
    in_var_alarmTime := var_timeAsDT,
    in_var_alarmCode1 := eP_alarmCode.GM,
    in_var_alarmCode2 := 5002,
    var_semaphore := var_semaphore,
    var_alarmQty := var_alarmQty,
    var_alarmListLog := var_alarmListLog,
    out_var_alarmListActive := gvl_error.var_ary_alarmlistActive); // fb_eventListGenerator

// NETWORK 43
fbi_eventListGenerator[41](
    in_flg_run := fun_setAlarm(in_flg_set := flg_errorTrg[41], in_flg_reset := gvl_error.flg_resetEventFlg),
    in_var_alarmTime := var_timeAsDT,
    var_semaphore := var_semaphore,
    var_alarmQty := var_alarmQty,
    var_alarmListLog := var_alarmListLog,
    out_var_alarmListActive := gvl_error.var_ary_alarmlistActive); // fb_eventListGenerator

// NETWORK 44
fbi_eventListGenerator[42](
    in_flg_run := fun_setAlarm(in_flg_set := flg_errorTrg[42], in_flg_reset := gvl_error.flg_resetEventFlg),
    in_var_alarmTime := var_timeAsDT,
    var_semaphore := var_semaphore,
    var_alarmQty := var_alarmQty,
    var_alarmListLog := var_alarmListLog,
    out_var_alarmListActive := gvl_error.var_ary_alarmlistActive); // fb_eventListGenerator

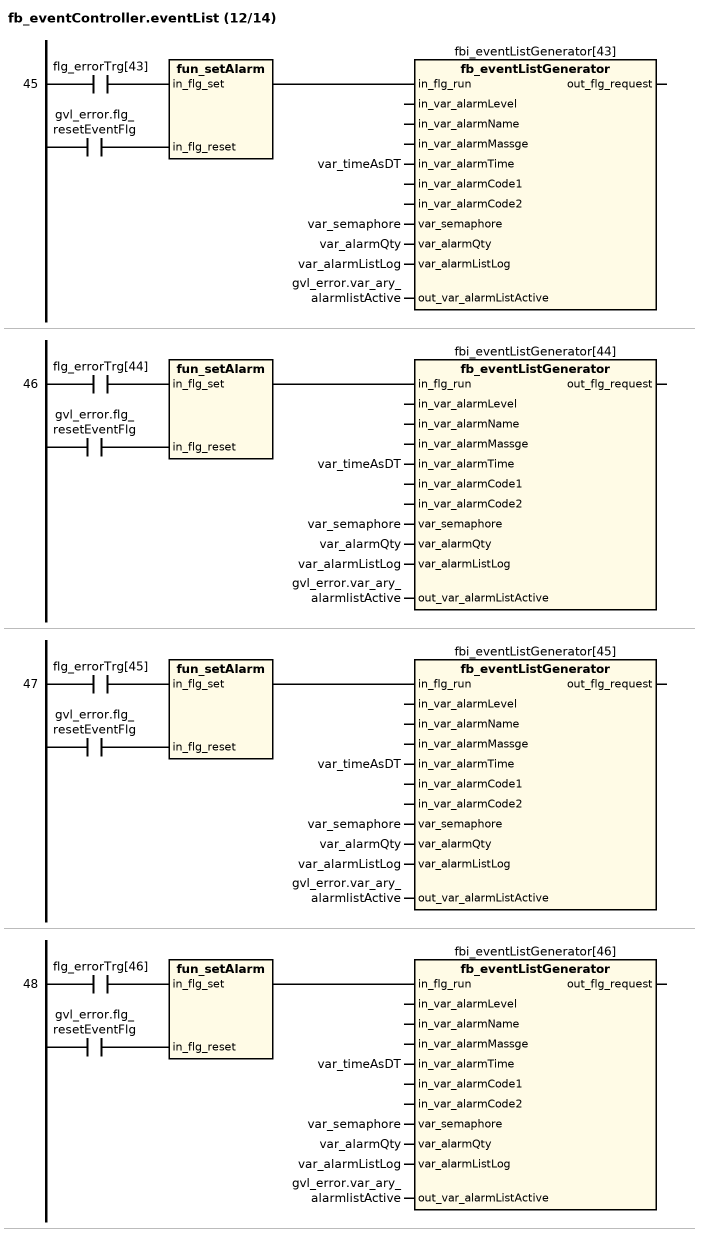
// NETWORK 45
fbi_eventListGenerator[43](
    in_flg_run := fun_setAlarm(in_flg_set := flg_errorTrg[43], in_flg_reset := gvl_error.flg_resetEventFlg),
    in_var_alarmTime := var_timeAsDT,
    var_semaphore := var_semaphore,
    var_alarmQty := var_alarmQty,
    var_alarmListLog := var_alarmListLog,
    out_var_alarmListActive := gvl_error.var_ary_alarmlistActive); // fb_eventListGenerator

// NETWORK 46
fbi_eventListGenerator[44](
    in_flg_run := fun_setAlarm(in_flg_set := flg_errorTrg[44], in_flg_reset := gvl_error.flg_resetEventFlg),
    in_var_alarmTime := var_timeAsDT,
    var_semaphore := var_semaphore,
    var_alarmQty := var_alarmQty,
    var_alarmListLog := var_alarmListLog,
    out_var_alarmListActive := gvl_error.var_ary_alarmlistActive); // fb_eventListGenerator

// NETWORK 47
fbi_eventListGenerator[45](
    in_flg_run := fun_setAlarm(in_flg_set := flg_errorTrg[45], in_flg_reset := gvl_error.flg_resetEventFlg),
    in_var_alarmTime := var_timeAsDT,
    var_semaphore := var_semaphore,
    var_alarmQty := var_alarmQty,
    var_alarmListLog := var_alarmListLog,
    out_var_alarmListActive := gvl_error.var_ary_alarmlistActive); // fb_eventListGenerator

// NETWORK 48
fbi_eventListGenerator[46](
    in_flg_run := fun_setAlarm(in_flg_set := flg_errorTrg[46], in_flg_reset := gvl_error.flg_resetEventFlg),
    in_var_alarmTime := var_timeAsDT,
    var_semaphore := var_semaphore,
    var_alarmQty := var_alarmQty,
    var_alarmListLog := var_alarmListLog,
    out_var_alarmListActive := gvl_error.var_ary_alarmlistActive); // fb_eventListGenerator

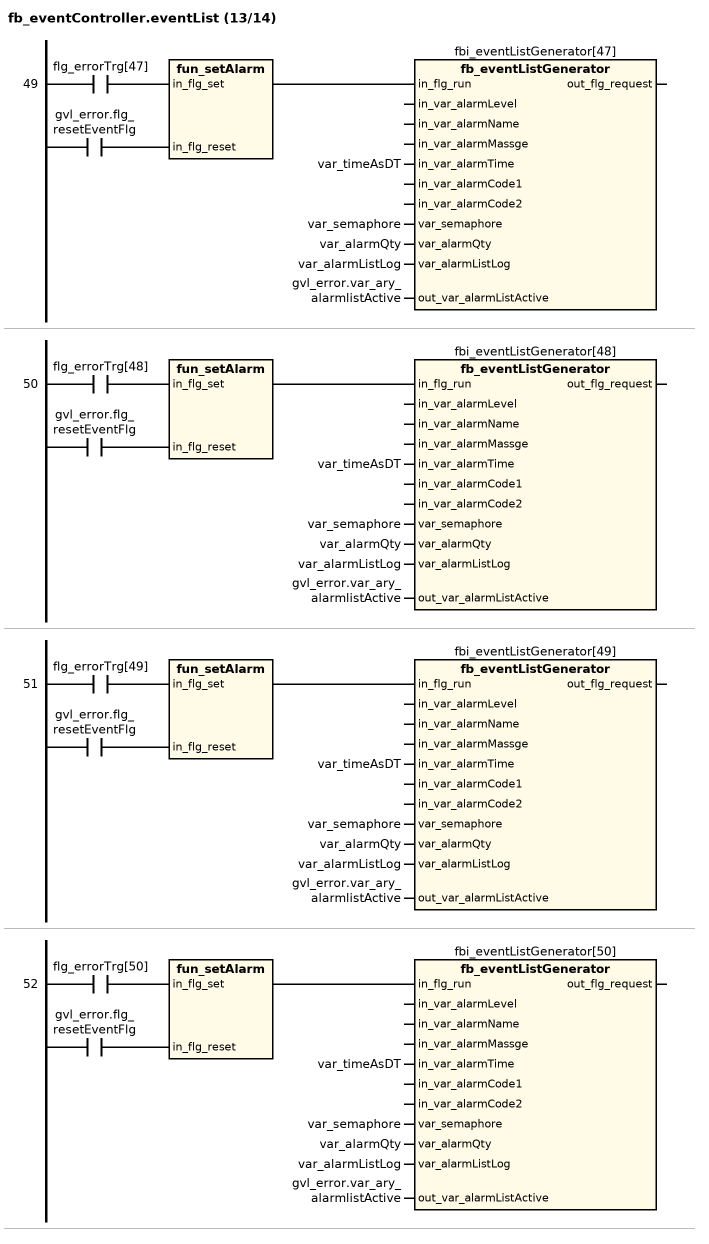
// NETWORK 49
fbi_eventListGenerator[47](
    in_flg_run := fun_setAlarm(in_flg_set := flg_errorTrg[47], in_flg_reset := gvl_error.flg_resetEventFlg),
    in_var_alarmTime := var_timeAsDT,
    var_semaphore := var_semaphore,
    var_alarmQty := var_alarmQty,
    var_alarmListLog := var_alarmListLog,
    out_var_alarmListActive := gvl_error.var_ary_alarmlistActive); // fb_eventListGenerator

// NETWORK 50
fbi_eventListGenerator[48](
    in_flg_run := fun_setAlarm(in_flg_set := flg_errorTrg[48], in_flg_reset := gvl_error.flg_resetEventFlg),
    in_var_alarmTime := var_timeAsDT,
    var_semaphore := var_semaphore,
    var_alarmQty := var_alarmQty,
    var_alarmListLog := var_alarmListLog,
    out_var_alarmListActive := gvl_error.var_ary_alarmlistActive); // fb_eventListGenerator

// NETWORK 51
fbi_eventListGenerator[49](
    in_flg_run := fun_setAlarm(in_flg_set := flg_errorTrg[49], in_flg_reset := gvl_error.flg_resetEventFlg),
    in_var_alarmTime := var_timeAsDT,
    var_semaphore := var_semaphore,
    var_alarmQty := var_alarmQty,
    var_alarmListLog := var_alarmListLog,
    out_var_alarmListActive := gvl_error.var_ary_alarmlistActive); // fb_eventListGenerator

// NETWORK 52
fbi_eventListGenerator[50](
    in_flg_run := fun_setAlarm(in_flg_set := flg_errorTrg[50], in_flg_reset := gvl_error.flg_resetEventFlg),
    in_var_alarmTime := var_timeAsDT,
    var_semaphore := var_semaphore,
    var_alarmQty := var_alarmQty,
    var_alarmListLog := var_alarmListLog,
    out_var_alarmListActive := gvl_error.var_ary_alarmlistActive); // fb_eventListGenerator

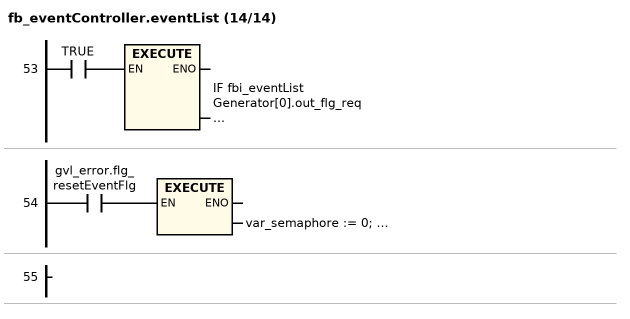
// NETWORK 53
IF fbi_eventListGenerator[0].out_flg_request OR
	fbi_eventListGenerator[1].out_flg_request OR
	fbi_eventListGenerator[2].out_flg_request OR
	fbi_eventListGenerator[3].out_flg_request OR
	fbi_eventListGenerator[4].out_flg_request OR
	fbi_eventListGenerator[5].out_flg_request OR
	fbi_eventListGenerator[6].out_flg_request OR
	fbi_eventListGenerator[7].out_flg_request OR
	fbi_eventListGenerator[8].out_flg_request OR
	fbi_eventListGenerator[9].out_flg_request OR
	fbi_eventListGenerator[10].out_flg_request OR
	fbi_eventListGenerator[11].out_flg_request OR
	fbi_eventListGenerator[12].out_flg_request OR
	fbi_eventListGenerator[13].out_flg_request OR
	fbi_eventListGenerator[14].out_flg_request OR
	fbi_eventListGenerator[15].out_flg_request OR
	fbi_eventListGenerator[16].out_flg_request OR
	fbi_eventListGenerator[17].out_flg_request OR
	fbi_eventListGenerator[18].out_flg_request OR
	fbi_eventListGenerator[19].out_flg_request OR
	fbi_eventListGenerator[20].out_flg_request OR
	fbi_eventListGenerator[21].out_flg_request OR
	fbi_eventListGenerator[22].out_flg_request OR
	fbi_eventListGenerator[23].out_flg_request OR
	fbi_eventListGenerator[24].out_flg_request OR
	fbi_eventListGenerator[25].out_flg_request OR
	fbi_eventListGenerator[26].out_flg_request OR
	fbi_eventListGenerator[27].out_flg_request OR
	fbi_eventListGenerator[28].out_flg_request OR
	fbi_eventListGenerator[29].out_flg_request OR
	fbi_eventListGenerator[30].out_flg_request OR
	fbi_eventListGenerator[31].out_flg_request OR
	fbi_eventListGenerator[32].out_flg_request OR
	fbi_eventListGenerator[33].out_flg_request OR
	fbi_eventListGenerator[34].out_flg_request OR
	fbi_eventListGenerator[35].out_flg_request OR
	fbi_eventListGenerator[36].out_flg_request OR
	fbi_eventListGenerator[37].out_flg_request OR
	fbi_eventListGenerator[38].out_flg_request OR
	fbi_eventListGenerator[39].out_flg_request OR
	fbi_eventListGenerator[40].out_flg_request OR
	fbi_eventListGenerator[41].out_flg_request OR
	fbi_eventListGenerator[42].out_flg_request OR
	fbi_eventListGenerator[43].out_flg_request OR
	fbi_eventListGenerator[44].out_flg_request OR
	fbi_eventListGenerator[44].out_flg_request OR
	fbi_eventListGenerator[45].out_flg_request OR
	fbi_eventListGenerator[46].out_flg_request OR
	fbi_eventListGenerator[47].out_flg_request OR
	fbi_eventListGenerator[48].out_flg_request OR
	fbi_eventListGenerator[49].out_flg_request OR
	fbi_eventListGenerator[50].out_flg_request THEN
		flg_reqUpdate := TRUE;
ELSE
	flg_reqUpdate := FALSE;
END_IF

// NETWORK 54
IF gvl_error.flg_resetEventFlg THEN
    var_semaphore := 0;
    var_alarmQty := 0;
END_IF

// NETWORK 55
END_ACTION

END_FUNCTION_BLOCK

(* stored: Version 1.1.0.1, ProductVersion 3.1.4024.11
   POU fb_eventController: Id {7bda6e1f-c0a6-402e-b5ac-c037b58a39f5}, SpecialFunc None
   Action eventList: Id {3397a22e-c581-44fa-bc2a-ac30fd56e34d} *)
